FUNCTION_BLOCK AX_TON (* Standard timer function block (on-delay timing) *)
  (* Standard: 61499-2; Classification: standard timer function block; Description: Copyright (c) 2024 HR Agrartechnik GmbH This program and the accompanying materials are made available under the terms of the Eclipse Public License 2.0 which is available at https://www.eclipse.org/legal/epl-2.0/ SPDX-License-Identifier: EPL-2.0 AX_TON -- On-delay timer FB with AX adapter interface The adapter input IN triggers execution (E1->REQ) and provides the boolean input value (D1->IN). The event input EIPT presets the delay time PT without triggering execution. When IN goes TRUE, Q becomes TRUE after delay PT. When IN goes FALSE, Q becomes FALSE immediately. *)
  (* Version 3.0, 2025-04-14, Patrick Aigner, changed package *)
  (* Version 1.0, 2024-03-04, Franz Höpfinger, HR Agrartechnik GmbH *)
  PACKAGE adapter::events::unidirectional::timers;
  IMPORT eclipse4diac::core::TypeHash;
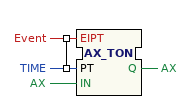
  EVENT_INPUT
    EIPT WITH PT; (* Set Preset Time (non-triggering) *)
  END_EVENT
  VAR_INPUT
    PT : TIME; (* Preset Time *)
  END_VAR
  SOCKETS
    IN : adapter::types::unidirectional::AX; (* Timer input (AX adapter) *)
  END_SOCKETS
  PLUGS
    Q : adapter::types::unidirectional::AX; (* Timer output (AX adapter) *)
  END_PLUGS
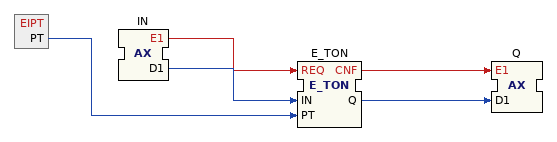
  FBS
    E_TON : iec61499::events::timers::E_TON;
  END_FBS
  EVENT_CONNECTIONS
    E_TON.CNF TO Q.E1;
    IN.E1 TO E_TON.REQ;
  END_CONNECTIONS
  DATA_CONNECTIONS
    E_TON.Q TO Q.D1;
    IN.D1 TO E_TON.IN;
    PT TO E_TON.PT;
  END_CONNECTIONS
END_FUNCTION_BLOCK
